(* IEC 61131-3 sources: ai-building-automation/docs/phase0/s1fix_evidence/run3/generated, 1 file *)

(* ---- PLC_PRG_decl.st ---- *)
PROGRAM PLC_PRG
VAR
    (* Deterministic demo for AHU-01 *)
    StartCommand : BOOL := FALSE;
    StopCommand : BOOL := FALSE;
    FanCommand : BOOL := FALSE;
    FanRunning : BOOL := FALSE;
    FanFault : BOOL := FALSE;
    SupplyTemp : REAL := 21.0;
    Setpoint : REAL := 22.0;
    FanSpeed : REAL := 50.0;
    HeatingValve : REAL := 0.0;
    (* Modbus TCP image (16-bit words, mapped to Modbus_TCP_Server I/O) *)
    Mb_Command : WORD; (* HR0 Command: bit0=StartCommand, bit1=StopCommand *)
    Mb_Status : WORD; (* IR0 Status: bit0=FanCommand, bit1=FanRunning, bit2=FanFault *)
END_VAR
